Staubli VAL3: RecordAlarm.pgx

program RecordAlarm()
  local string l_sString
  local joint l_jJoint
begin
  if !$fileExists("Log://alarm.txt")
    nFileID=$fileOpen("Log://alarm.txt","w")
  else
    nFileID=$fileOpen("Log://alarm.txt","a")
  endIf



  if nFileID<0 or nFileID>9
    return
  endIf

  l_sString=getDate("%Y_%m_%d %H:%M:%S")
  l_sString=l_sString+"急停触发:产品:"+DataBase:sProductName[DataBase:nWorkPlaceIndex]+"路径:"+toString("",DataBase:nTrajIndex)
  l_sString=l_sString+"MoveID:"+toString(".3",getMoveId())

  $fileSet(nFileID,l_sString,1)
  l_jJoint=herej()

  l_sString="关节位置:"+toString(".3",l_jJoint.j1)+","+toString(".3",l_jJoint.j2)+","+toString(".3",l_jJoint.j3)+","
  l_sString= l_sString+toString(".3",l_jJoint.j4)+","+toString(".3",l_jJoint.j5)+","+toString(".3",l_jJoint.j6)

   $fileSet(nFileID,l_sString,1)

   $fileClose(nFileID)









end
